// TIA Portal V19 export
TYPE "OOAx_Alr"
// stored: Access Published
   STRUCT
      TargetPosIncorrect : Bool;   // Target position is out of limit range
      PosOutTolerance : Bool;   // Position out of tolerance
      WrongDirection : Bool;
      WrongNotIncrease : Bool;
      HwLimitMinus : Bool;
      HwLimitPlus : Bool;
      TimeoutPreset : Bool;
   END_STRUCT;
END_TYPE
